SUBAPPLICATION Softkey_Aux_Switch_Auto_TO_Remote_WRITE (* VT-SoftKey lesen ODER AUX-Zuweisung (Joystick) lesen ODER lokaler Web-Override ODER ein zusaetzlicher physischer Taster auf einem ANDEREN Modul (Remote-Subscribe) ODER Automatik-Kommando + Remote-OPC-UA-Write an Zielmodul (generisch, ein Kanal, ohne Status-Feedback) - 5-Quellen-Erweiterung von Softkey_Aux_Switch_TO_Remote_WRITE um einen zusaetzlichen AUTO_IN-Socket (z.B. Befuellautomatik-Hysterese, die dieselbe Fuellband-Heben-Leitung ansteuert wie SoftKey/AUX/Web/physischer Taster S08). *)
  (* Standard: 61499-2; Description: Copyright (c) 2026 Meisterschulen am Ostbahnhof This program and the accompanying materials are made available under the terms of the Eclipse Public License 2.0 which is available at https://www.eclipse.org/legal/epl-2.0/ SPDX-License-Identifier: EPL-2.0 *)
  (* Version 1.2, 2026-09-27, Franz Höpfinger, Meisterschulen am Ostbahnhof, Franz: 'die Automatik muss auch ausschalten wenn man das Fuellband manuell hebt, sonst faengt der Bunkerboden an zu laufen wenn man ueber die Schwelle kommt' - neuer Plug MANUAL_OUT (NUR SoftKey/Aux/Web/Switch, OHNE Automatik-Anteil - sonst wuerde die Automatik sich durch ihr eigenes Kommando selbst abschalten). OR_MERGE (AX_OR_5) aufgeteilt in OR_Manual (AX_OR_4, die 4 manuellen Quellen) + OR_Automatik (AX_OR_2, OR_Manual ODER AUTO_IN) - unveraendertes Gesamtverhalten fuer CMD_OUT/Remote-Write. *)
  (* Version 1.0, 2026-09-13, Franz Höpfinger, Meisterschulen am Ostbahnhof, initial implementation - 5-Quellen-Variante von Softkey_Aux_Switch_TO_Remote_WRITE (AX_OR_5 statt AX_OR_4, zusaetzlicher AUTO_IN-Socket), fuer Fuellband Heben (Befuellautomatik-Hysterese zusaetzlich zu SoftKey/AUX/Web/physischem Taster S08). *)
  PACKAGE MyLib::sys;
  IMPORT isobus::UT::Q::const::IDs::ID_NULL;
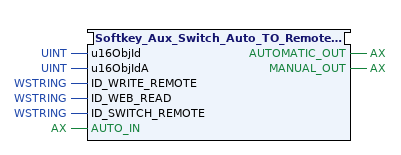
  VAR_INPUT
    u16ObjId : UINT := ID_NULL; (* Object ID SoftKey (VT) *)
    u16ObjIdA : UINT := ID_NULL; (* Object ID AuxFunction2 (VT) *)
    ID_WRITE_REMOTE : WSTRING; (* Remote-Write-Adresse zum Zielmodul (Befehl, ACTION=WRITE, CLIENT) *)
    ID_WEB_READ : WSTRING; (* Lokale Subscribe-Adresse fuer einen Web-Client (z.B. vt-ui-mirror) auf demselben Modul, ODER-verknuepft mit SoftKey und AUX *)
    ID_SWITCH_REMOTE : WSTRING; (* Remote-Subscribe-Adresse eines zusaetzlichen physischen Tasters auf einem ANDEREN Modul, ODER-verknuepft mit SoftKey/AUX/Web/Automatik *)
  END_VAR
  SOCKETS
    AUTO_IN : adapter::types::unidirectional::AX; (* Autonomes Kommando (z.B. Befuellautomatik-Hysterese), ODER-verknuepft mit SoftKey/Aux/Web/physischem Taster *)
  END_SOCKETS
  PLUGS
    AUTOMATIC_OUT : adapter::types::unidirectional::AX; (* Optional: lokal gemergter Rohbefehl (SoftKey ODER AUX ODER Web ODER Switch ODER Automatik), VOR dem Remote-Write - unverdrahtet lassen, wenn nicht gebraucht *)
    MANUAL_OUT : adapter::types::unidirectional::AX; (* Optional: NUR die manuellen Quellen (SoftKey ODER AUX ODER Web ODER Switch), OHNE AUTO_IN - z.B. um eine Automatik abzuschalten, wenn der Bediener manuell eingreift, ohne dass sich die Automatik durch ihr eigenes Kommando selbst abschaltet. Unverdrahtet lassen, wenn nicht gebraucht. *)
  END_PLUGS
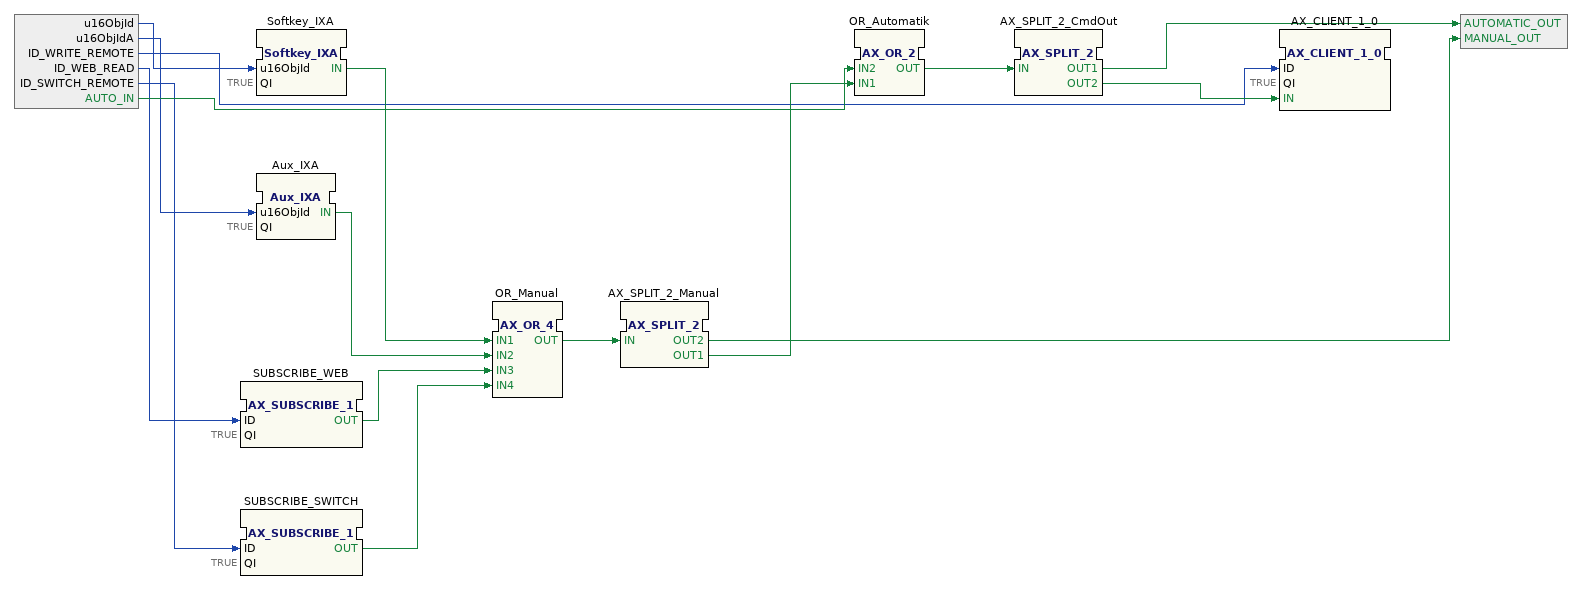
  FBS
    Softkey_IXA : isobus::UT::io::Softkey::Softkey_IXA(QI := TRUE);
    Aux_IXA : isobus::UT::io::Auxiliary::IN::Aux_IXA(QI := TRUE);
    SUBSCRIBE_WEB : adapter::net::AX_SUBSCRIBE_1(QI := TRUE);
    SUBSCRIBE_SWITCH : adapter::net::AX_SUBSCRIBE_1(QI := TRUE);
    OR_Manual : adapter::booleanOperators::AX_OR_4;
    AX_SPLIT_2_Manual : adapter::events::unidirectional::AX_SPLIT_2;
    OR_Automatik : adapter::booleanOperators::AX_OR_2;
    AX_CLIENT_1_0 : adapter::net::AX_CLIENT_1_0(QI := TRUE);
    AX_SPLIT_2_CmdOut : adapter::events::unidirectional::AX_SPLIT_2;
  END_FBS
  DATA_CONNECTIONS
    u16ObjId TO Softkey_IXA.u16ObjId;
    u16ObjIdA TO Aux_IXA.u16ObjId;
    ID_WEB_READ TO SUBSCRIBE_WEB.ID;
    ID_SWITCH_REMOTE TO SUBSCRIBE_SWITCH.ID;
    ID_WRITE_REMOTE TO AX_CLIENT_1_0.ID;
  END_CONNECTIONS
  ADAPTER_CONNECTIONS
    Softkey_IXA.IN TO OR_Manual.IN1;
    Aux_IXA.IN TO OR_Manual.IN2;
    SUBSCRIBE_WEB.OUT TO OR_Manual.IN3;
    SUBSCRIBE_SWITCH.OUT TO OR_Manual.IN4;
    OR_Manual.OUT TO AX_SPLIT_2_Manual.IN;
    AX_SPLIT_2_Manual.OUT2 TO MANUAL_OUT;
    AUTO_IN TO OR_Automatik.IN2;
    OR_Automatik.OUT TO AX_SPLIT_2_CmdOut.IN;
    AX_SPLIT_2_CmdOut.OUT1 TO AUTOMATIC_OUT;
    AX_SPLIT_2_CmdOut.OUT2 TO AX_CLIENT_1_0.IN;
    AX_SPLIT_2_Manual.OUT1 TO OR_Automatik.IN1;
  END_CONNECTIONS
END_SUBAPPLICATION
